{attribute addProperty BoxType "ELX9560-0000-0018"}
{attribute addProperty Id "Uin_OKAT %I*BOOL81"}
{attribute addProperty CRC "1363173712"}
{attribute addProperty SizeInBites "8"}
{attribute addProperty SizeInBytes "1"}
TYPE Status_Uin_51406150 :
STRUCT
	{attribute addProperty Name "Uin_OK"}
	Uin_OK AT %I* : BOOL;
END_STRUCT
END_TYPE

(* stored: Version 1.2.0.0, ProductVersion 3.1.4024.9
   DUT Status_Uin_51406150: Id {c1688f96-7db2-49da-8886-bb3082377738} *)
